ADAPTER CompoundAdapterWith (* Adapter with events and data, not all data WITHed *)
  (* Standard: 61499-1; Description: Copyright (c) 2023 Johannes Kepler University Linz This program and the accompanying materials are made available under the terms of the Eclipse Public License 2.0 which is available at https://www.eclipse.org/legal/epl-2.0/ SPDX-License-Identifier: EPL-2.0 *)
  (* Version 1.0, 2023-03-08, Bianca Wiesmayr, Johannes Kepler University Linz, initial API and implementation and/or initial documentation *)
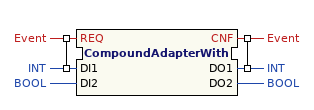
  EVENT_INPUT
    REQ WITH DI1; (* Request from Socket *)
  END_EVENT
  EVENT_OUTPUT
    CNF WITH DO1; (* Confirmation from Plug *)
  END_EVENT
  VAR_INPUT
    DI1 : INT := 42;
    DI2 : BOOL := TRUE;
  END_VAR
  VAR_OUTPUT
    DO1 : INT := 21;
    DO2 : BOOL;
  END_VAR
END_ADAPTER
